// TIA Portal V17 export
// export: Created 2022-06-27T13:57:05.9331622Z, ExportSetting WithDefaults, DisplayName Totally Integrated Automation Portal, DisplayVersion V17 Update 3, DisplayName TIA Portal Openness, DisplayVersion V17 Update 3, DisplayName TIA Portal Version Control Interface, DisplayVersion V17, DisplayName SINAMICS Startdrive Advanced, DisplayVersion V17 Update1, DisplayName SINAMICS Startdrive G110M, G120, G120C, G120D, G120P, G115D, DisplayVersion V17 Update1, DisplayName SINAMICS Startdrive G130, G150, S120, S150, SINAMICS MV, S210, DisplayVersion V17 Update1, DisplayName STEP 7 Professional, DisplayVersion V17 Update 3, DisplayName STEP 7 Safety, DisplayVersion V17, DisplayName WinCC UA Professional, DisplayVersion V17 Update 3
FUNCTION_BLOCK "S031_ONOFF_VALVES"   // FB31, LAD
{ S7_Optimized_Access := 'TRUE' }
VERSION : 0.1
// stored: AutoNumber false, IsIECCheckEnabled false, IsRetainMemResEnabled false, MemoryReserve 100, SetENOAutomatically false, UDAEnableTagReadback false
BEGIN

REGION Network 2: FV26-3B - Chamber 1 Feeder - Automatic on and off
END_REGION

REGION Network 3: FV26-3B - Chamber 1 Feeder - Interlocks
END_REGION

REGION Network 4: FV26-3B - Chamber 1 Feeder - Valve Function Call
END_REGION

REGION Network 6: FV26-4C - Chamber 1 Discharge - Automatic on and off
END_REGION

REGION Network 7: FV26-4C - Chamber 1 Discharge - Interlocks
END_REGION

REGION Network 8: FV26-4C - Chamber 1 Discharge - Valve Function Call
END_REGION

REGION Network 10: FV26-4B - Cooler 1 Discharge - Automatic on and off
END_REGION

REGION Network 11: FV26-4B - Cooler 1 Discharge - Interlocks
END_REGION

REGION Network 12: FV26-4B - Cooler 1 Discharge - Valve Function Call
END_REGION

REGION Network 14: FV26-5C - Fan Valve Roaster to Chamber 2 - Automatic on and off
END_REGION

REGION Network 15: FV26-5C - Fan Valve Roaster to Chamber 2 - Interlocks
END_REGION

REGION Network 16: FV26-5C - Fan Valve Roaster to Chamber 2 - Valve Function Call
END_REGION

REGION Network 18: FV26-5B - Fan Valve Dryer to Chamber 1 - Automatic on and off
END_REGION

REGION Network 19: FV26-5B - Fan Valve Dryer to Chamber 1 - Interlocks
END_REGION

REGION Network 20: FV26-5B - Fan Valve Dryer to Chamber 1 - Valve Function Call
END_REGION

REGION Network 22: FV26-6C - Fan Branch Valve Cooler - Automatic on and off
END_REGION

REGION Network 23: FV26-6C - Fan Branch Valve Cooler - Interlocks
END_REGION

REGION Network 24: FV26-6C - Fan Branch Valve Cooler - Valve Function Call
END_REGION

REGION Network 26: FV26-6B - Cooler 2 Discharge - Automatic on and off
END_REGION

REGION Network 27: FV26-6B - Cooler 2 Discharge - Interlocks
END_REGION

REGION Network 28: FV26-6B - Cooler 2 Discharge - Valve Function Call
END_REGION

REGION Network 30: FV26-7C - Chamber 2 Discharge - Automatic on and off
END_REGION

REGION Network 31: FV26-7C - Chamber 2 Discharge - Interlocks
END_REGION

REGION Network 32: FV26-7C - Chamber 2 Discharge - Valve Function Call
END_REGION

REGION Network 34: FV26-7B - Chamber 2 Feeder - Automatic on and off
END_REGION

REGION Network 35: FV26-7B - Chamber 2 Feeder - Interlocks
END_REGION

REGION Network 36: FV26-7B - Chamber 2 Feeder - Valve Function Call
END_REGION

REGION Network 38: FV26-8C - Branch Valve Manual Bagging / Regular Transport - Automatic on and off
END_REGION

REGION Network 39: FV26-8C - Branch Valve Manual Bagging / Regular Transport - Interlocks
END_REGION

REGION Network 40: FV26-8C - Branch Valve Manual Bagging / Regular Transport - Valve Function Call
END_REGION

REGION Network 42: FV26-8B - Branch Valve Manual Bagging / Regular Transport - Automatic on and off
END_REGION

REGION Network 43: FV26-8B - Branch Valve Manual Bagging / Regular Transport - Interlocks
END_REGION

REGION Network 44: FV26-8B - Branch Valve Manual Bagging / Regular Transport - Valve Function Call
END_REGION

REGION Network 46: FV26-9C - Spare - Automatic on and off
END_REGION

REGION Network 47: FV26-9C - Spare - Interlocks
END_REGION

REGION Network 48: FV26-9C - Spare - Valve Function Call
END_REGION
END_FUNCTION_BLOCK
